{attribute 'GeneratedUsingTerminal: AT2050-0501-0020'}
{attribute addProperty BoxType "AT2050-0501-0020"}
{attribute addProperty Id "A_0087_AT2050_5501_0016_AT2050_5501AT2050_01D6DEDF80"}
{attribute addProperty CRC "996865047"}
{attribute addProperty Size "80"}
TYPE A_0057_AT2050_0501_0020_3B6AF417 EXTENDS AT2050_86175B41 :
STRUCT
	{attribute addProperty Name "A_0087_AT2050_5501_0016_AT2050_5501"}
	{attribute addProperty PreviousPort "A_0057(AT2050-0501-0020) : B"}
	A_0087_AT2050_5501_0016_AT2050_5501 : AT2050_01D6DEDF;
END_STRUCT
END_TYPE

(* stored: Version 1.2.0.0, ProductVersion 3.1.4024.9
   DUT A_0057_AT2050_0501_0020_3B6AF417: Id {c65ae2d6-75a9-4afb-bbfe-eeba9f46e5c6} *)
